PROGRAM prgHouse
VAR
	fbKBusState					: FB_K_Bus_State;
	uint_KBusState				: UINT;							//{#lynus.ag#()}
	lrHousePower				: LREAL;								//{#lynus.ag#()}
	lrNetzEinspeisung			: LREAL;								//{#lynus.ag#()}
	lrBetriebMuellerBau			: LREAL;								//{#lynus.ag#()}
	lrElektromobilitaet			: LREAL;								//{#lynus.ag#()}
	lrHolzschnitzel				: LREAL;								//{#lynus.ag#()}
	lrLueftung_Kaelte			: LREAL;								//{#lynus.ag#()}
	rPVProd						: REAL;									//{#lynus.ag#()}
	lrAbgaenge					: REAL;									//{#lynus.ag#()}
	fbGrid1						: FB_EM_Beckhoff_KL3403;  	//Elektromobilität 
	fbGrid2						: FB_EM_Beckhoff_KL3403;	//Holzschnitzelheizung
	fbGrid3						: FB_EM_Beckhoff_KL3403;	//Lüftung/Kälte Büro
	
	

    Volt1L1  AT %I* : REAL;
    Strom1L1 AT %I* : REAL;
	//UV Müller Holzbau
	ActivePowerTotal_1	AT %I*	: REAL;									//{#lynus.ag#()}
	//Abgang Direktmessung
	ActivePowerTotal_2	AT %I*	: REAL;									//{#lynus.ag#()}
	//Produktion PV
	ActivePowerTotal_3	AT %I*	: REAL;									//{#lynus.ag#()}

END_VAR

lrNetzEinspeisung := ActivePowerTotal_1/1000 + ActivePowerTotal_2/1000 - rPVProd;

lrElektromobilitaet	:= fbGrid1.stDataEMPower.lrPowerTotal;
lrHolzschnitzel		:= fbGrid2.stDataEMPower.lrPowerTotal;
lrLueftung_Kaelte	:= fbGrid3.stDataEMPower.lrPowerTotal;
lrHousePower		:= ActivePowerTotal_1/1000 + fbGrid1.stDataEMPower.lrPowerTotal + fbGrid2.stDataEMPower.lrPowerTotal + fbGrid3.stDataEMPower.lrPowerTotal;

lrBetriebMuellerBau := -fbGrid1.stDataEMPower.lrPowerTotal - fbGrid2.stDataEMPower.lrPowerTotal - fbGrid3.stDataEMPower.lrPowerTotal + lrHousePower;	

rPVProd				:= (ActivePowerTotal_3)/100 * -1;					//Invertieren
lrAbgaenge 			:= ActivePowerTotal_2/1000;
//lrHousePower 		:= lrBetriebMuellerBau * -1;						//Invertierte Einspeisung für Darstellung

//The mapping of this function must be linked with the K-Bus State in the E/A Part
fbKBusState(	uiKBusState_OUT=> , 
				b_Kbus_notOk=> , 
				word_ErrorCount=> );

fbGrid1(
	bEnable:= TRUE, 
	bChannel1Invers:= FALSE, 
	bChannel2Invers:= FALSE, 
	bChannel3Invers:= FALSE, 
	uiCurrentTransformerRatioL1:= 400, 
	uiCurrentTransformerRatioL2:= 400, 
	uiCurrentTransformerRatioL3:= 400, 
	uiKBusState_IN:= fbKBusState.uiKBusState_OUT, 
	stDataEMPower=> , 
	stDataEMCounter=> , 
	stDataEMPowerRealTime=> , 
	stDataEMCounterRealTime=> , 
	diNrOfEM_OUT=> );
	
	
fbGrid2(
	bEnable:= TRUE, 
	bChannel1Invers:= FALSE, 
	bChannel2Invers:= FALSE, 
	bChannel3Invers:= FALSE, 
	uiCurrentTransformerRatioL1:= 400, 
	uiCurrentTransformerRatioL2:= 400, 
	uiCurrentTransformerRatioL3:= 400, 
	uiKBusState_IN:= , 
	stDataEMPower=> , 
	stDataEMCounter=> , 
	stDataEMPowerRealTime=> , 
	stDataEMCounterRealTime=> , 
	diNrOfEM_OUT=> );
	
fbGrid3(
	bEnable:= TRUE, 
	bChannel1Invers:= FALSE, 
	bChannel2Invers:= FALSE, 
	bChannel3Invers:= FALSE, 
	uiCurrentTransformerRatioL1:= 400, 
	uiCurrentTransformerRatioL2:= 400, 
	uiCurrentTransformerRatioL3:= 400, 
	uiKBusState_IN:= , 
	stDataEMPower=> , 
	stDataEMCounter=> , 
	stDataEMPowerRealTime=> , 
	stDataEMCounterRealTime=> , 
	diNrOfEM_OUT=> );

END_PROGRAM

(* stored: Version 1.1.0.1, ProductVersion 3.1.4024.13
   POU prgHouse: Id {2627c3a1-fabe-46fd-8396-cc823b8dfb91}, SpecialFunc None *)
